// TIA Portal V19 export
FUNCTION_BLOCK "Mixer_Block"   // FB3, LAD
TITLE = Control of Mixer Unit
{ S7_Optimized_Access := 'TRUE' }
// Simple Mixer Design and Animation
// stored: MemoryReserve 100, SetENOAutomatically false
BEGIN

REGION Network 1: Start Mixer
   // Turns Mixer On , Refreshes at 2Hz for Animation.
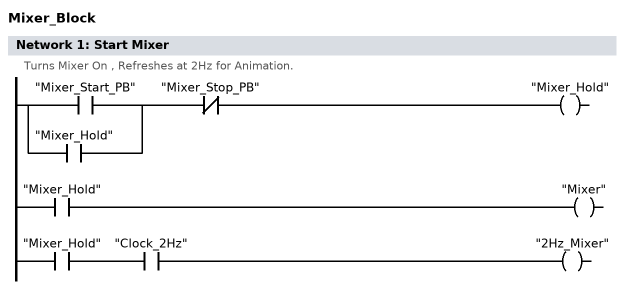
   RUNG wire#powerrail
      Contact( "Mixer_Start_PB" )
      wire#w1
      I_Contact( "Mixer_Stop_PB" )
      Coil( "Mixer_Hold" )
   END_RUNG
   RUNG wire#powerrail
      Contact( "Mixer_Hold" )
   END_RUNG wire#w1
   RUNG wire#powerrail
      Contact( "Mixer_Hold" )
      Coil( "Mixer" )
   END_RUNG
   RUNG wire#powerrail
      Contact( "Mixer_Hold" )
      Contact( "Clock_2Hz" )
      Coil( "2Hz_Mixer" )
   END_RUNG
   // the same network as SCL:
   "Mixer_Hold" := ("Mixer_Start_PB" OR "Mixer_Hold") AND NOT "Mixer_Stop_PB";
   "Mixer" := "Mixer_Hold";
   "2Hz_Mixer" := "Mixer_Hold" AND "Clock_2Hz";
END_REGION
END_FUNCTION_BLOCK
